{attribute 'linkalways'} 
{attribute 'no_explicit_call' := 'This FB is a CLASS and must be accessed using methods or properties'}
{attribute 'enable_dynamic_creation'}
FUNCTION_BLOCK Node_F_VN_GaussianFilterExp EXTENDS VisionNode
VAR
	ipSrcImage : _ITcVnImage;
    ipDestImage : _ITcVnImage;
    nFilterWidth : _UDINT(1);
    nFilterHeight : _UDINT(1);
    fSigmaX : _LREAL(0.0);
    fSigmaY : _LREAL(0.0);
    eBorderType : _ETcVnBorderInterpolationMethod(ETcVnBorderInterpolationMethod.TCVN_BIM_DEFAULT);
    hrPrev : _HRESULT(S_OK);
	hresult : _HRESULT(S_OK);
END_VAR

METHOD PUBLIC  Clone : I_Node
VAR
	pNode : POINTER TO Node_F_VN_GaussianFilterExp;
END_VAR
pNode := __NEW(Node_F_VN_GaussianFilterExp);
Clone := pNode^;
END_METHOD

METHOD FB_init : BOOL
VAR_INPUT
	bInitRetains : BOOL; // if TRUE, the retain variables are initialized (warm start / cold start)
	bInCopyCode : BOOL;  // if TRUE, the instance afterwards gets moved into the copy code (online change)
END_VAR
AddInput('ipSrcImage', ipSrcImage);
AddParameter('nFilterWidth', nFilterWidth);
AddParameter('nFilterHeight', nFilterHeight);
AddParameter('fSigmaX', fSigmaX);
AddParameter('fSigmaY', fSigmaY);
AddParameter('eBorderType', eBorderType);
AddInput('hrPrev', hrPrev);
AddOutput('ipDestImage', ipDestImage);
AddOutput('hresult',hresult);
END_METHOD

METHOD PROTECTED OnExecute
hresult.Value := F_VN_GaussianFilterExp(
	ipSrcImage := ipSrcImage.Value,
	ipDestImage := ipDestImage.Value,
	nFilterWidth := nFilterWidth.Value,
	nFilterHeight := nFilterHeight.Value,
    fSigmaX := fSigmaX.Value,
    fSigmaY := fSigmaY.Value,
    eBorderType := eBorderType.Value,
	hrPrev := hrPrev.Value);
END_METHOD

METHOD PUBLIC PreExecutionCheck
VAR_INPUT
	Check : I_PreExecutionChecks;
END_VAR
Check.IsTrue(ipSrcImage.IsValid, 'ipSrcImage must contain an image');
Check.IsTrue(nFilterWidth.IsOdd, 'nFilterWidth must be an odd number');
Check.IsTrue(nFilterHeight.IsOdd, 'nFilterHeight must be an odd number');
Check.IsTrue((fSigmaX.Value >= 0), 'fSigmaX must be greater than or equal to 0');
Check.IsTrue((fSigmaY.Value >= 0), 'fSigmaY must be greater than or equal to 0');
END_METHOD

END_FUNCTION_BLOCK

(* stored: Version 1.1.0.1, ProductVersion 3.1.4024.15
   POU Node_F_VN_GaussianFilterExp: Id {7a70e77e-3100-0441-1ec5-05e1b18f4581}, SpecialFunc None
   Folder Constructor: Id {97ba2879-3db2-0421-11a4-f95ee5638170}
   Method Clone: Id {e085c6ef-7166-080d-3c8b-84b055dcf803}
   Method FB_init: Id {a06a42fe-9184-00a5-11b2-a65d7671a8e4}
   Method OnExecute: Id {64cf7006-36c6-02bf-23ff-7e11019527c1}
   Method PreExecutionCheck: Id {32c0e213-a803-0d93-2102-d0d8d2f0924c} *)
